Staubli VAL3: JointTrajPtMsg.dtx

public Header header
  [0]
    num nMsgType
    num nCommType
    num nReplyCode
    num nData[12]
public JointTrajPt jointTrajPt
  [0]
    num nSeq
    num nJoints[10]
    num nVelocity
    num nDuration
public Prefix prefix
  [0]
    num nLength
    num nData[4]
public Body body
  [0]
    num nData[64]
